// TIA Portal V16 export
// export: Created 2022-07-21T09:35:29.4881636Z, ExportSetting WithDefaults, DisplayName Totally Integrated Automation Portal, DisplayVersion V16 Update 4, DisplayName TIA Portal Version Control Interface, DisplayVersion V16 Update 2, DisplayName TIA Portal Openness, DisplayVersion V16 Update 4, DisplayName SINAMICS Startdrive Advanced, DisplayVersion V16 Update 5, DisplayName SINAMICS Startdrive G130, G150, S120, S150, SINAMICS MV, S210, DisplayVersion V16 Update 5, DisplayName SINAMICS Startdrive G110M, G120, G120C, G120D, G120P, G115D, DisplayVersion V16 Update 5, DisplayName STEP 7 Professional, DisplayVersion V16 Update 4, DisplayName STEP 7 Safety, DisplayVersion V16, DisplayName WinCC Advanced, DisplayVersion V16 Update 4
FUNCTION_BLOCK "fbInterrollCnv"   // FB213, LAD
TITLE = Interroll conveyor handling / Obsługa przenośnika Interroll
{ S7_Optimized_Access := 'TRUE' }
AUTHOR : a32thzz
VERSION : 0.1
// stored: AutoNumber true, IsIECCheckEnabled false, IsRetainMemResEnabled false, MemoryReserve 100, SetENOAutomatically false, UDAEnableTagReadback false
   VAR_INPUT
      disableAlarms : Bool;
      dataFromSafety : Bool;
      blockedZone : Bool;   // Blokowanie ruchu podczas przejazdu przez czujnik / Block movement during transfer through sensor
      startTPDelayTime : DInt;   // Opóźnienie rozpoczęcia przejazdu przez czujnik / Delay start transfer through sensor
      group : "typeGroup";
   END_VAR
   VAR_IN_OUT
      data : "typeInterrollUniversalFullCnvDrive";
   END_VAR
   VAR
      autoStart : Bool;
      delayPTAlm0 : Time := T#5s;   // Czas opóźnienia dla alarmu 0 / delay alarm 0
      delayPTAlm1 : Time := T#1s;   // Czas opóźnienia dla alarmu 1 / delay alarm 1
      delayPTAlm2 : Time := T#1s;   // Czas opóźnienia dla alarmu 2 / delay alarm 2
      delayPTAlm3 : Time := T#1s;   // Czas opóźnienia dla alarmu 3 / delay alarm 3
      delayPTAlm4 : Time := T#1s;   // Czas opóźnienia dla alarmu 4 / delay alarm 4
      delayPTAlm5 : Time := T#1s;   // Czas opóźnienia dla alarmu 5 / delay alarm 5
      delayPTAlm6 : Time := T#1s;   // Czas opóźnienia dla alarmu 7 / delay alarm 7
      delayPTAlm7 : Time := T#1s;   // Czas opóźnienia dla alarmu 6 / delay alarm 6
      instTmrDlyAlm0 { S7_SetPoint := 'True'} : TON_TIME;   // Opóźnienie dla alarmu 0 / delay alarm 0
      instTmrDlyAlm1 { S7_SetPoint := 'True'} : TON_TIME;   // Opóźnienie dla alarmu 1 / delay alarm 1
      instTmrDlyAlm2 { S7_SetPoint := 'True'} : TON_TIME;   // Opóźnienie dla alarmu 2 / delay alarm 2
      instTmrDlyAlm3 { S7_SetPoint := 'True'} : TON_TIME;   // Opóźnienie dla alarmu 3 / delay alarm 3
      instTmrDlyAlm4 { S7_SetPoint := 'True'} : TON_TIME;   // Opóźnienie dla alarmu 4 / delay alarm 4
      instTmrDlyAlm5 { S7_SetPoint := 'True'} : TON_TIME;   // Opóźnienie dla alarmu 5 / delay alarm 5
      instTmrDlyAlm6 { S7_SetPoint := 'True'} : TON_TIME;   // Opóźnienie dla alarmu 7 / delay alarm 7
      instTmrDlyAlm7 { S7_SetPoint := 'True'} : TON_TIME;   // Opóźnienie dla alarmu 6 / delay alarm 6
      instTmrOnDlySensor1 { S7_SetPoint := 'True'} : TON_TIME;
      statStartMoveDelay { ExternalAccessible := 'False'; ExternalVisible := 'False'; ExternalWritable := 'False'} : Bool;
   END_VAR
   VAR_TEMP
      bAlm0 : Bool;   // tymczasowy bit alarmu 0 / temporary alarm bit 0
      bAlm1 : Bool;   // tymczasowy bit alarmu 1 / temporary alarm bit 1
      bAlm2 : Bool;   // tymczasowy bit alarmu 2 / temporary alarm bit 2
      bAlm3 : Bool;   // tymczasowy bit alarmu 3 / temporary alarm bit 3
      bAlm4 : Bool;   // tymczasowy bit alarmu 4 / temporary alarm bit 4
      bAlm5 : Bool;   // tymczasowy bit alarmu 5 / temporary alarm bit 5
      bAlm6 : Bool;   // tymczasowy bit alarmu 6 / temporary alarm bit 6
      bAlm7 : Bool;   // tymczasowy bit alarmu 7 / temporary alarm bit 7
   END_VAR
   VAR_TEMP   // added for the SCL form of the ladder/FBD networks
      _w1 : Bool;
   END_VAR
BEGIN

REGION Network 1: Alarm: Drive error (while power on) / Alarm: Błąd napędu (przy załączonym zasilaniu)
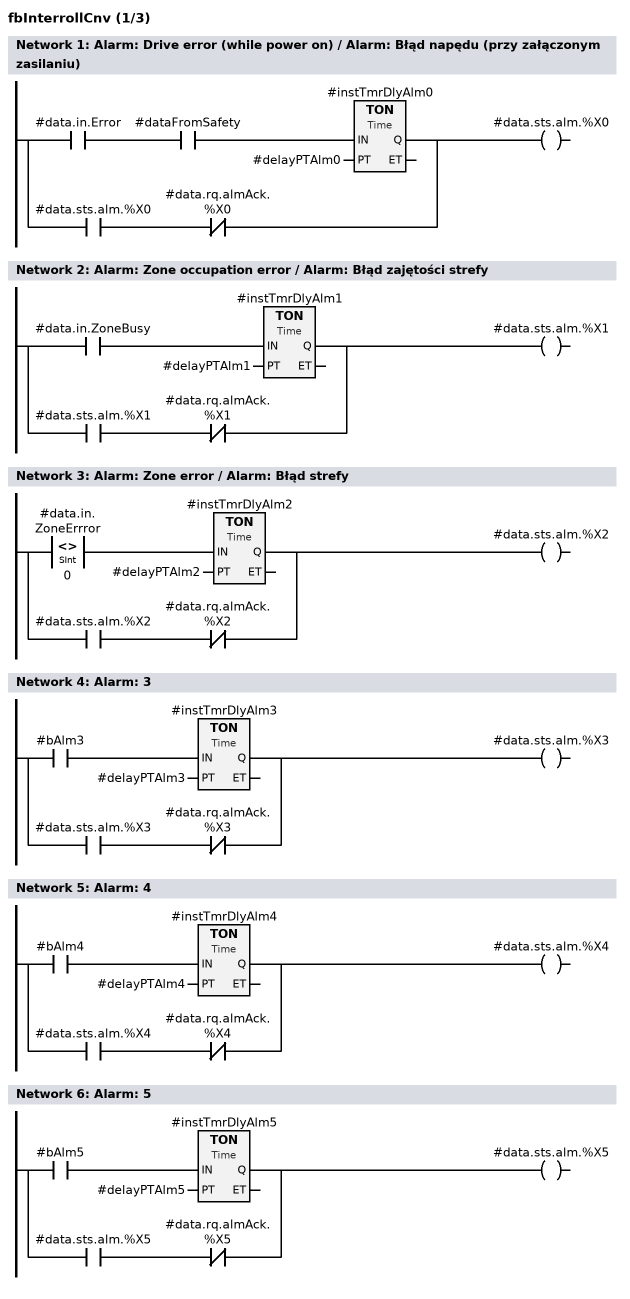
   RUNG wire#powerrail
      Contact( #data.in.Error )
      Contact( #dataFromSafety )
      { S7_Templates := "time_type := Time" } #instTmrDlyAlm0.TON(pt := #delayPTAlm0, et =>)
      wire#w1
      Coil( #data.sts.alm.%X0 )
   END_RUNG
   RUNG wire#powerrail
      Contact( #data.sts.alm.%X0 )
      I_Contact( #data.rq.almAck.%X0 )
   END_RUNG wire#w1
   // the same network as SCL:
   #instTmrDlyAlm0(IN := #data.in.Error AND #dataFromSafety, PT := #delayPTAlm0);   // TON
   #data.sts.alm.%X0 := #instTmrDlyAlm0.Q OR (#data.sts.alm.%X0 AND NOT #data.rq.almAck.%X0);
END_REGION

REGION Network 2: Alarm: Zone occupation error / Alarm: Błąd zajętości strefy
   RUNG wire#powerrail
      Contact( #data.in.ZoneBusy )
      { S7_Templates := "time_type := Time" } #instTmrDlyAlm1.TON(pt := #delayPTAlm1, et =>)
      wire#w1
      Coil( #data.sts.alm.%X1 )
   END_RUNG
   RUNG wire#powerrail
      Contact( #data.sts.alm.%X1 )
      I_Contact( #data.rq.almAck.%X1 )
   END_RUNG wire#w1
   // the same network as SCL:
   #instTmrDlyAlm1(IN := #data.in.ZoneBusy, PT := #delayPTAlm1);   // TON
   #data.sts.alm.%X1 := #instTmrDlyAlm1.Q OR (#data.sts.alm.%X1 AND NOT #data.rq.almAck.%X1);
END_REGION

REGION Network 3: Alarm: Zone error / Alarm: Błąd strefy
   RUNG wire#powerrail
      { S7_Templates := "SrcType := SInt" } NE_Contact(in1 := #data.in.ZoneErrror, in2 := 0)
      { S7_Templates := "time_type := Time" } #instTmrDlyAlm2.TON(pt := #delayPTAlm2, et =>)
      wire#w1
      Coil( #data.sts.alm.%X2 )
   END_RUNG
   RUNG wire#powerrail
      Contact( #data.sts.alm.%X2 )
      I_Contact( #data.rq.almAck.%X2 )
   END_RUNG wire#w1
   // the same network as SCL:
   #instTmrDlyAlm2(IN := #data.in.ZoneErrror <> 0, PT := #delayPTAlm2);   // TON
   #data.sts.alm.%X2 := #instTmrDlyAlm2.Q OR (#data.sts.alm.%X2 AND NOT #data.rq.almAck.%X2);
END_REGION

REGION Network 4: Alarm: 3
   RUNG wire#powerrail
      Contact( #bAlm3 )
      { S7_Templates := "time_type := Time" } #instTmrDlyAlm3.TON(pt := #delayPTAlm3, et =>)
      wire#w1
      Coil( #data.sts.alm.%X3 )
   END_RUNG
   RUNG wire#powerrail
      Contact( #data.sts.alm.%X3 )
      I_Contact( #data.rq.almAck.%X3 )
   END_RUNG wire#w1
   // the same network as SCL:
   #instTmrDlyAlm3(IN := #bAlm3, PT := #delayPTAlm3);   // TON
   #data.sts.alm.%X3 := #instTmrDlyAlm3.Q OR (#data.sts.alm.%X3 AND NOT #data.rq.almAck.%X3);
END_REGION

REGION Network 5: Alarm: 4
   RUNG wire#powerrail
      Contact( #bAlm4 )
      { S7_Templates := "time_type := Time" } #instTmrDlyAlm4.TON(pt := #delayPTAlm4, et =>)
      wire#w1
      Coil( #data.sts.alm.%X4 )
   END_RUNG
   RUNG wire#powerrail
      Contact( #data.sts.alm.%X4 )
      I_Contact( #data.rq.almAck.%X4 )
   END_RUNG wire#w1
   // the same network as SCL:
   #instTmrDlyAlm4(IN := #bAlm4, PT := #delayPTAlm4);   // TON
   #data.sts.alm.%X4 := #instTmrDlyAlm4.Q OR (#data.sts.alm.%X4 AND NOT #data.rq.almAck.%X4);
END_REGION

REGION Network 6: Alarm: 5
   RUNG wire#powerrail
      Contact( #bAlm5 )
      { S7_Templates := "time_type := Time" } #instTmrDlyAlm5.TON(pt := #delayPTAlm5, et =>)
      wire#w1
      Coil( #data.sts.alm.%X5 )
   END_RUNG
   RUNG wire#powerrail
      Contact( #data.sts.alm.%X5 )
      I_Contact( #data.rq.almAck.%X5 )
   END_RUNG wire#w1
   // the same network as SCL:
   #instTmrDlyAlm5(IN := #bAlm5, PT := #delayPTAlm5);   // TON
   #data.sts.alm.%X5 := #instTmrDlyAlm5.Q OR (#data.sts.alm.%X5 AND NOT #data.rq.almAck.%X5);
END_REGION

REGION Network 7: Alarm: 6
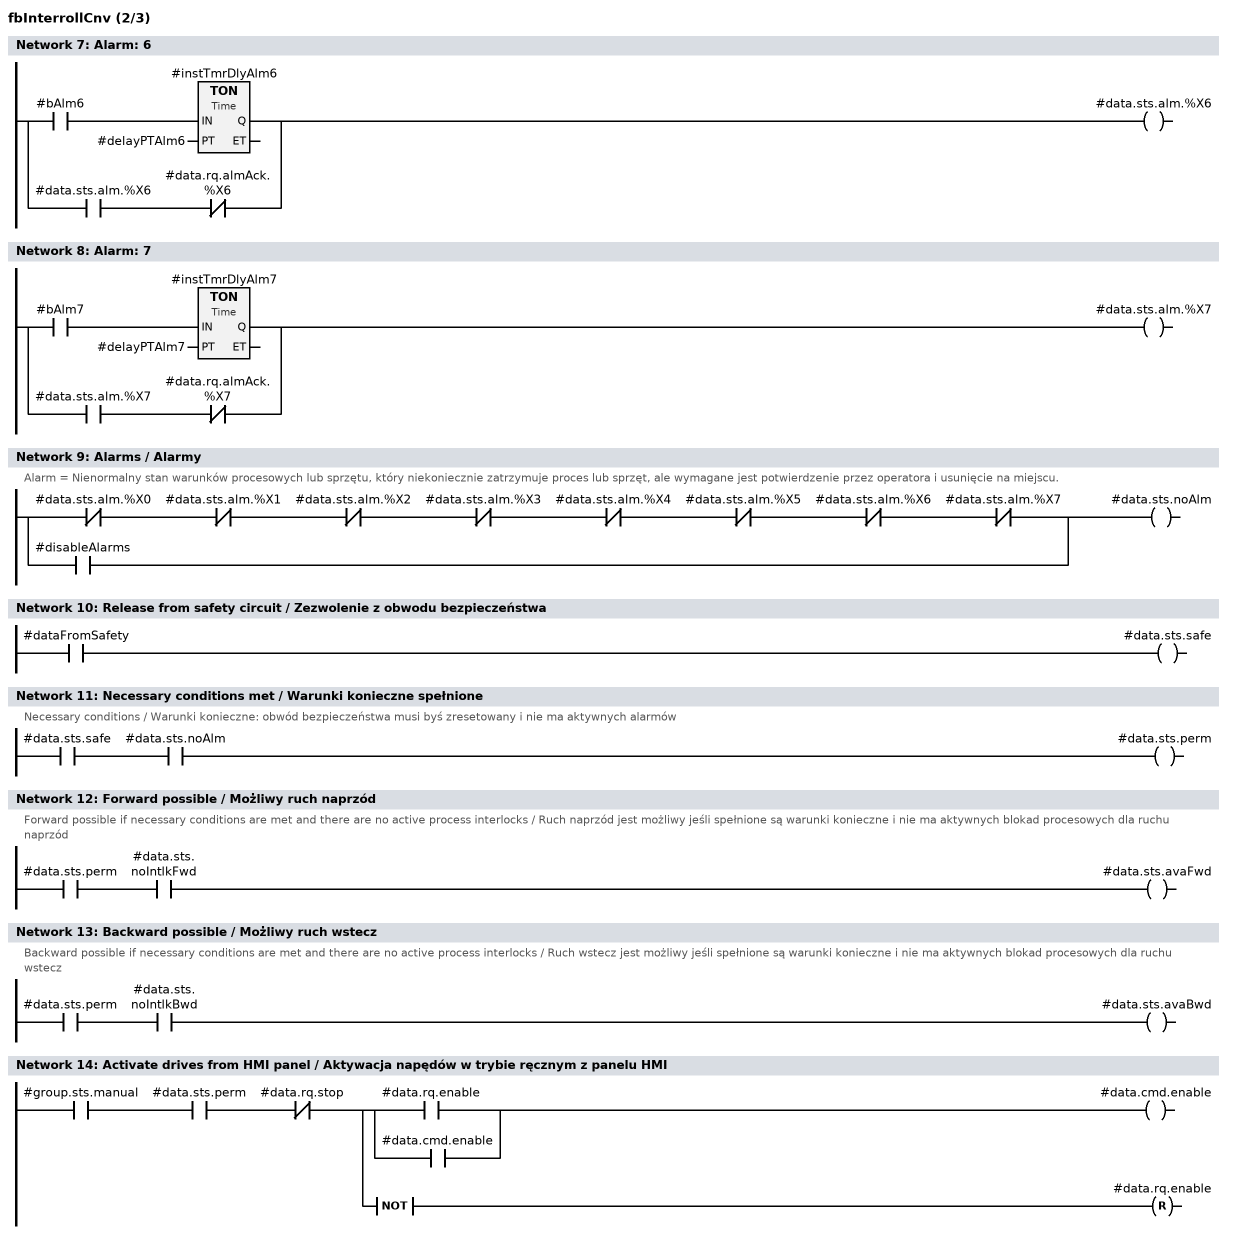
   RUNG wire#powerrail
      Contact( #bAlm6 )
      { S7_Templates := "time_type := Time" } #instTmrDlyAlm6.TON(pt := #delayPTAlm6, et =>)
      wire#w1
      Coil( #data.sts.alm.%X6 )
   END_RUNG
   RUNG wire#powerrail
      Contact( #data.sts.alm.%X6 )
      I_Contact( #data.rq.almAck.%X6 )
   END_RUNG wire#w1
   // the same network as SCL:
   #instTmrDlyAlm6(IN := #bAlm6, PT := #delayPTAlm6);   // TON
   #data.sts.alm.%X6 := #instTmrDlyAlm6.Q OR (#data.sts.alm.%X6 AND NOT #data.rq.almAck.%X6);
END_REGION

REGION Network 8: Alarm: 7
   RUNG wire#powerrail
      Contact( #bAlm7 )
      { S7_Templates := "time_type := Time" } #instTmrDlyAlm7.TON(pt := #delayPTAlm7, et =>)
      wire#w1
      Coil( #data.sts.alm.%X7 )
   END_RUNG
   RUNG wire#powerrail
      Contact( #data.sts.alm.%X7 )
      I_Contact( #data.rq.almAck.%X7 )
   END_RUNG wire#w1
   // the same network as SCL:
   #instTmrDlyAlm7(IN := #bAlm7, PT := #delayPTAlm7);   // TON
   #data.sts.alm.%X7 := #instTmrDlyAlm7.Q OR (#data.sts.alm.%X7 AND NOT #data.rq.almAck.%X7);
END_REGION

REGION Network 9: Alarms / Alarmy
   // Alarm = Nienormalny stan warunków procesowych lub sprzętu, który niekoniecznie zatrzymuje proces lub sprzęt, ale wymagane jest potwierdzenie przez operatora i usunięcie na miejscu.
   RUNG wire#powerrail
      I_Contact( #data.sts.alm.%X0 )
      I_Contact( #data.sts.alm.%X1 )
      I_Contact( #data.sts.alm.%X2 )
      I_Contact( #data.sts.alm.%X3 )
      I_Contact( #data.sts.alm.%X4 )
      I_Contact( #data.sts.alm.%X5 )
      I_Contact( #data.sts.alm.%X6 )
      I_Contact( #data.sts.alm.%X7 )
      wire#w1
      Coil( #data.sts.noAlm )
   END_RUNG
   RUNG wire#powerrail
      Contact( #disableAlarms )
   END_RUNG wire#w1
   // the same network as SCL:
   #data.sts.noAlm := (NOT #data.sts.alm.%X0 AND NOT #data.sts.alm.%X1 AND NOT #data.sts.alm.%X2 AND NOT #data.sts.alm.%X3 AND NOT #data.sts.alm.%X4 AND NOT #data.sts.alm.%X5 AND NOT #data.sts.alm.%X6 AND NOT #data.sts.alm.%X7) OR #disableAlarms;
END_REGION

REGION Network 10: Release from safety circuit / Zezwolenie z obwodu bezpieczeństwa
   RUNG wire#powerrail
      Contact( #dataFromSafety )
      Coil( #data.sts.safe )
   END_RUNG
   // the same network as SCL:
   #data.sts.safe := #dataFromSafety;
END_REGION

REGION Network 11: Necessary conditions met / Warunki konieczne spełnione
   // Necessary conditions / Warunki konieczne: obwód bezpieczeństwa musi byś zresetowany i nie ma aktywnych alarmów
   RUNG wire#powerrail
      Contact( #data.sts.safe )
      Contact( #data.sts.noAlm )
      Coil( #data.sts.perm )
   END_RUNG
   // the same network as SCL:
   #data.sts.perm := #data.sts.safe AND #data.sts.noAlm;
END_REGION

REGION Network 12: Forward possible / Możliwy ruch naprzód
   // Forward possible if necessary conditions are met and there are no active process interlocks / Ruch naprzód jest możliwy jeśli spełnione są warunki konieczne i nie ma aktywnych blokad procesowych dla ruchu naprzód
   RUNG wire#powerrail
      Contact( #data.sts.perm )
      Contact( #data.sts.noIntlkFwd )
      Coil( #data.sts.avaFwd )
   END_RUNG
   // the same network as SCL:
   #data.sts.avaFwd := #data.sts.perm AND #data.sts.noIntlkFwd;
END_REGION

REGION Network 13: Backward possible / Możliwy ruch wstecz
   // Backward possible if necessary conditions are met and there are no active process interlocks / Ruch wstecz jest możliwy jeśli spełnione są warunki konieczne i nie ma aktywnych blokad procesowych dla ruchu wstecz
   RUNG wire#powerrail
      Contact( #data.sts.perm )
      Contact( #data.sts.noIntlkBwd )
      Coil( #data.sts.avaBwd )
   END_RUNG
   // the same network as SCL:
   #data.sts.avaBwd := #data.sts.perm AND #data.sts.noIntlkBwd;
END_REGION

REGION Network 14: Activate drives from HMI panel / Aktywacja napędów w trybie ręcznym z panelu HMI
   RUNG wire#powerrail
      Contact( #group.sts.manual )
      Contact( #data.sts.perm )
      I_Contact( #data.rq.stop )
      wire#w1
      Contact( #data.rq.enable )
      wire#w2
      Coil( #data.cmd.enable )
   END_RUNG
   RUNG wire#w1
      Contact( #data.cmd.enable )
   END_RUNG wire#w2
   RUNG wire#w1
      Not()
      R_Coil( #data.rq.enable )
   END_RUNG
   // the same network as SCL:
   #_w1 := #group.sts.manual AND #data.sts.perm AND NOT #data.rq.stop;
   #data.cmd.enable := #_w1 AND (#data.rq.enable OR #data.cmd.enable);
   IF NOT #_w1 THEN #data.rq.enable := FALSE; END_IF;
END_REGION

REGION Network 15: Enable axis / Załącz oś
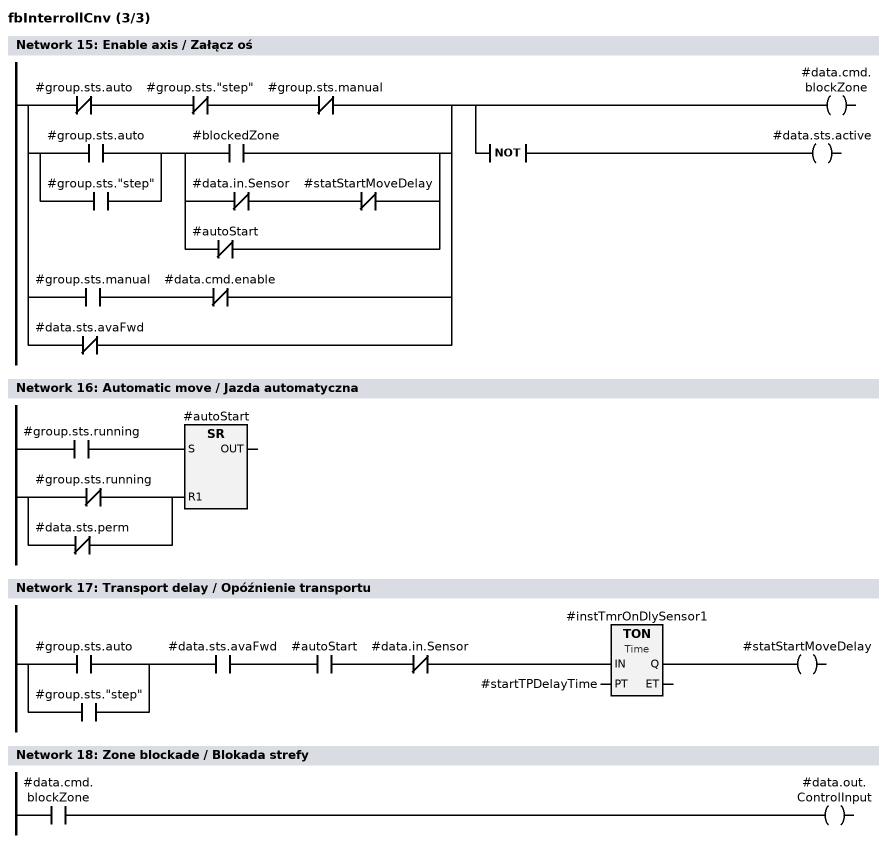
   RUNG wire#powerrail
      I_Contact( #group.sts.auto )
      I_Contact( #group.sts."step" )
      I_Contact( #group.sts.manual )
      wire#w1
      Coil( #data.cmd.blockZone )
   END_RUNG
   RUNG wire#powerrail
      Contact( #group.sts.auto )
      wire#w2
      Contact( #blockedZone )
   END_RUNG wire#w1
   RUNG wire#powerrail
      Contact( #group.sts."step" )
   END_RUNG wire#w2
   RUNG wire#w2
      I_Contact( #data.in.Sensor )
      I_Contact( #statStartMoveDelay )
   END_RUNG wire#w1
   RUNG wire#w2
      I_Contact( #autoStart )
   END_RUNG wire#w1
   RUNG wire#powerrail
      Contact( #group.sts.manual )
      I_Contact( #data.cmd.enable )
   END_RUNG wire#w1
   RUNG wire#powerrail
      I_Contact( #data.sts.avaFwd )
   END_RUNG wire#w1
   RUNG wire#w1
      Not()
      Coil( #data.sts.active )
   END_RUNG
   // the same network as SCL:
   #data.cmd.blockZone := (NOT #group.sts.auto AND NOT #group.sts."step" AND NOT #group.sts.manual) OR ((#group.sts.auto OR #group.sts."step") AND (#blockedZone OR (NOT #data.in.Sensor AND NOT #statStartMoveDelay) OR NOT #autoStart)) OR (#group.sts.manual AND NOT #data.cmd.enable) OR NOT #data.sts.avaFwd;
   #data.sts.active := NOT #data.cmd.blockZone;
END_REGION

REGION Network 16: Automatic move / Jazda automatyczna
   RUNG wire#powerrail
      Contact( #group.sts.running )
      S_SR(operand := #autoStart, r1 := wire#w1)
   END_RUNG
   RUNG wire#powerrail
      I_Contact( #group.sts.running )
   END_RUNG wire#w1
   RUNG wire#powerrail
      I_Contact( #data.sts.perm )
   END_RUNG wire#w1
   // the same network as SCL:
   IF #group.sts.running THEN
       #autoStart := TRUE;   // SR flip-flop
   END_IF;
   IF NOT #group.sts.running OR NOT #data.sts.perm THEN #autoStart := FALSE; END_IF;
END_REGION

REGION Network 17: Transport delay / Opóźnienie transportu
   RUNG wire#powerrail
      Contact( #group.sts.auto )
      wire#w1
      Contact( #data.sts.avaFwd )
      Contact( #autoStart )
      I_Contact( #data.in.Sensor )
      { S7_Templates := "time_type := Time" } #instTmrOnDlySensor1.TON(pt := #startTPDelayTime, et =>)
      Coil( #statStartMoveDelay )
   END_RUNG
   RUNG wire#powerrail
      Contact( #group.sts."step" )
   END_RUNG wire#w1
   // the same network as SCL:
   #instTmrOnDlySensor1(IN := (#group.sts.auto OR #group.sts."step") AND #data.sts.avaFwd AND #autoStart AND NOT #data.in.Sensor,   // TON
                        PT := #startTPDelayTime);
   #statStartMoveDelay := #instTmrOnDlySensor1.Q;
END_REGION

REGION Network 18: Zone blockade / Blokada strefy
   RUNG wire#powerrail
      Contact( #data.cmd.blockZone )
      Coil( #data.out.ControlInput )
   END_RUNG
   // the same network as SCL:
   #data.out.ControlInput := #data.cmd.blockZone;
END_REGION
END_FUNCTION_BLOCK
